Universal Robots PolyScope program: Main_JF.urp

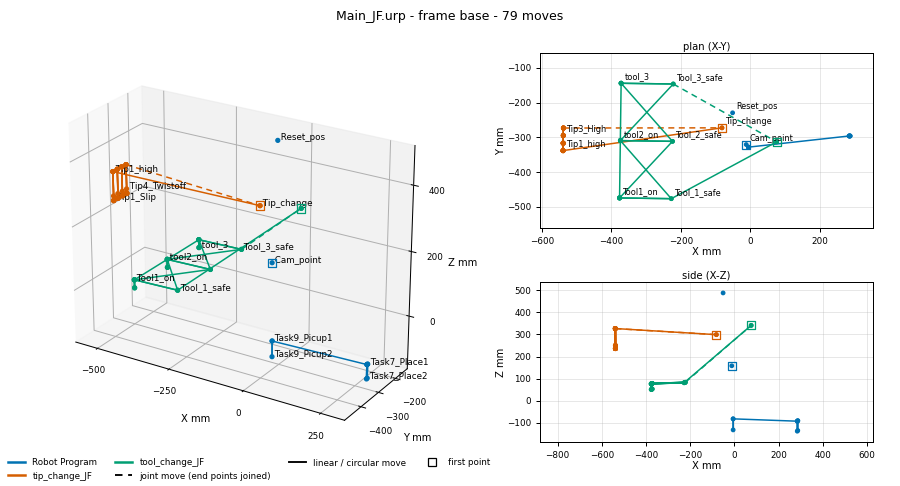
[picture p0: tool path of Main_JF.urp in frame base, 79 of 86 moves have a stored position in this frame; points joined in program order, loops and branches not executed]
Program Main_JF (installation=default directory=/programs/usbdisk/Billeder fra kamera createdIn=3.7.0.40195 lastSavedIn=3.10.1.76190 robotSerialNumber=2018359886)
Calibrated DH parameters: a=[-0.000111, -0.180064, -0.391564, 0.000025, 0.000035, 0]; d=[0.089308, 162.079685, -160.155007, -1.814221, 0.094754, 0.082578]; alpha=[1.569707, -0.002379, 0.010338, 1.570474, -1.569894, 0]; deltaTheta=[0.000021, -1.133914, 1.184629, -0.050828, 0.000017, 0.000075]
BeforeStart
  open := socket_open("192.168.0.15",30002)
  Old_Tool := 0
  Old_tip := 0
  Set DigitalOutput pin=config_out[4]; digitalValue=0
  Set DigitalOutput pin=config_out[5]; digitalValue=0
  Set DigitalOutput pin=config_out[6]; digitalValue=0
  Set DigitalOutput pin=config_out[7]; digitalValue=0
  Set DigitalOutput pin=config_out[0]; digitalValue=1
  Set DigitalOutput pin=config_out[2]; digitalValue=1
  Call Tool_initiation_tjeck
Robot Program (runOnlyOnce=false)
  Loop While (checkContinuously=false) expression=open≟ False
    open := socket_open("192.168.0.15",30002)
    Wait Sleep waitTime=0.5
  data := socket_read_ascii_float(8)
  Wait Sleep waitTime=0.5
  If data[0]≠0
    task := data[1]
    New_Tool_Setup := data[2]
    X_axis := data[3]
    Y_axis := data[4]
    Z_axis := data[5]
    X_rot := data[6]
    Y_rot := data[7]
    Z_rot := data[8]
    Rot := [d2r(data[6]),d2r(data[7]),d2r(data[8])]
    rot_v := rpy2rotvec(Rot)
    Insect_pos_High := p[X_axis,Y_axis,Z_axis+0.05,rot_v[0],rot_v[1],rot_v[2]]
    Insect_pos := p[X_axis,Y_axis,Z_axis,rot_v[0],rot_v[1],rot_v[2]]
    If New_Tool_Setup≠0
      If New_Tool_Setup>3
        New_tip := New_Tool_Setup-1
        New_Tool := 1
        Set NoAction tcp=TCP_Tips
      Else 
        New_tip := 0
        New_Tool := New_Tool_Setup
    Else 
      New_Tool := 0
      New_tip := 0
    If Old_Tool≟1 and New_tip≠Old_tip
      Call tip_change_JF
    SuppressedNode
      Switch expression=New_Tool
        Case (caseValue=1)
          Set NoAction tcp=TCP_Tool1
        Case (caseValue=2)
          Set NoAction tcp=TCP_Tool2
        Case (caseValue=3)
          Set NoAction tcp=TCP_Tool3
    If New_Tool≠Old_Tool
      Call tool_change_JF
    If New_tip≠Old_tip
      Call tip_change_JF
    SuppressedNode
      If New_tip≠Old_tip
        Popup Message (haltProgram=false message=Mount the correct tool tip. inputType=Text)
        Old_tip := New_tip
    If task≟1
      Wait Sleep waitTime=0.5
      Set SingleDigitalPulseActionState SingleDigitalPulseActionState(hiPulseInSeconds=0.5, pin=config_out[4])
      Set SingleDigitalPulseActionState SingleDigitalPulseActionState(hiPulseInSeconds=0.5, pin=config_out[5])
      Set SingleDigitalPulseActionState SingleDigitalPulseActionState(hiPulseInSeconds=0.5, pin=config_out[6])
      Set SingleDigitalPulseActionState SingleDigitalPulseActionState(hiPulseInSeconds=0.5, pin=config_out[7])
      Wait AnalogInput pin=analog_in[0]; analogComparison=0; analogValue=4
      Wait Sleep waitTime=0.5
      MoveL speed 250 mm/s, acceleration 1200 mm/s^2 (useActiveTCP=false) tcp=TCP_Cam; feature=Base
        SuppressedNode
          Waypoint ST_0_pos: TCP in base x=-75.138 y=-256.156 z=-140.441 mm, rx=0.4782 ry=3.0882 rz=0.0296 rad; joints [-83.913, -73.866, -152.197, -44.779, -268.413, 24.148] deg; flange x=-80.553 y=-258.226 z=132.545 mm, rx=0.4782 ry=3.0882 rz=0.0296 rad
        Waypoint Cam_point: TCP in base x=-11.711 y=-320.976 z=158.38 mm, rx=-0.0005 ry=-0.0003 rz=-3.1411 rad; joints [-100.01, -73.764, -127.296, -67.748, 91.294, -10.022] deg; flange x=-166.479 y=-319.785 z=277.387 mm, rx=-0.0077 ry=3.1318 rz=-0.0369 rad
        Wait Sleep waitTime=12
        SuppressedNode
          Waypoint Waypoint_1 (Relative): TCP in base x=286.294 y=-286.187 z=165.302 mm, rx=-0.0004 ry=0.0004 rz=3.1278 rad; joints [-44.345, -64.751, -131.64, -72.299, -270.032, 46.416] deg; flange x=131.485 y=-282.783 z=284.213 mm, rx=0.0146 ry=3.1313 rz=-0.0371 rad
    If task≟2
      Wait Sleep waitTime=0.5
      Set SingleDigitalPulseActionState SingleDigitalPulseActionState(hiPulseInSeconds=0.5, pin=config_out[4])
      Set SingleDigitalPulseActionState SingleDigitalPulseActionState(hiPulseInSeconds=0.5, pin=config_out[5])
      Set SingleDigitalPulseActionState SingleDigitalPulseActionState(hiPulseInSeconds=0.5, pin=config_out[6])
      Set SingleDigitalPulseActionState SingleDigitalPulseActionState(hiPulseInSeconds=0.5, pin=config_out[7])
      Wait AnalogInput pin=analog_in[0]; analogComparison=0; analogValue=4
      Wait Sleep waitTime=0.5
    If task≟3
      Wait Sleep waitTime=0.5
      Set SingleDigitalPulseActionState SingleDigitalPulseActionState(hiPulseInSeconds=0.5, pin=config_out[6])
      Set SingleDigitalPulseActionState SingleDigitalPulseActionState(hiPulseInSeconds=0.5, pin=config_out[7])
      Wait AnalogInput pin=analog_in[0]; analogComparison=0; analogValue=4
      Wait Sleep waitTime=0.5
    If task≟4
      Wait Sleep waitTime=0.5
      Set SingleDigitalPulseActionState SingleDigitalPulseActionState(hiPulseInSeconds=0.5, pin=config_out[4])
      Set SingleDigitalPulseActionState SingleDigitalPulseActionState(hiPulseInSeconds=0.5, pin=config_out[6])
      Set SingleDigitalPulseActionState SingleDigitalPulseActionState(hiPulseInSeconds=0.5, pin=config_out[7])
      Wait AnalogInput pin=analog_in[0]; analogComparison=0; analogValue=4
      Wait Sleep waitTime=0.5
    If task≟5
      Wait Sleep waitTime=0.5
      Set SingleDigitalPulseActionState SingleDigitalPulseActionState(hiPulseInSeconds=0.5, pin=config_out[5])
      Set SingleDigitalPulseActionState SingleDigitalPulseActionState(hiPulseInSeconds=0.5, pin=config_out[6])
      Set SingleDigitalPulseActionState SingleDigitalPulseActionState(hiPulseInSeconds=0.5, pin=config_out[7])
      Wait AnalogInput pin=analog_in[0]; analogComparison=0; analogValue=4
      Wait Sleep waitTime=0.5
    If task≟6
      Wait Sleep waitTime=0.5
      Set SingleDigitalPulseActionState SingleDigitalPulseActionState(hiPulseInSeconds=0.5, pin=config_out[4])
      Wait AnalogInput pin=analog_in[0]; analogComparison=0; analogValue=4
      Wait Sleep waitTime=0.5
      Set SingleDigitalPulseActionState SingleDigitalPulseActionState(hiPulseInSeconds=0.5, pin=config_out[5])
      Wait AnalogInput pin=analog_in[0]; analogComparison=0; analogValue=4
      Wait Sleep waitTime=0.5
    If task≟7
      Wait Sleep waitTime=0.5
      If New_Tool_Setup≟1
        Set NoAction tcp=TCP_Tool1
      Else 
        Set NoAction tcp=TCP_Tips
      MoveL speed 250 mm/s, acceleration 1200 mm/s^2 (useActiveTCP=true) feature=Base
        SuppressedNode
          Waypoint Task7_Picup1: TCP in base x=-2.957 y=-327.485 z=-88.615 mm, rx=-0.0002 ry=-0.0001 rz=1.5744 rad; joints [-84.172, -77.712, -147.228, -41.841, -255.532, 22.481] deg; flange x=-59.467 y=-294.342 z=154.237 mm, rx=0.3968 ry=2.8622 rz=0.009 rad
        SuppressedNode
          Waypoint Task7_Picup2: TCP in base x=-2.9 y=-327.528 z=-136.598 mm, rx=-0.0002 ry=0 rz=1.5745 rad; joints [-84.173, -87.531, -150.911, -28.32, -255.654, 22.544] deg; flange x=-59.407 y=-294.371 z=106.252 mm, rx=0.3967 ry=2.8623 rz=0.0089 rad
        Waypoint Waypoint (Variable): variable=Insect_pos_High
        SuppressedNode
          Waypoint Waypoint (Variable): variable=Insect_pos
      Set SingleDigitalPulseActionState SingleDigitalPulseActionState(hiPulseInSeconds=0.5, pin=config_out[6])
      Wait AnalogInput pin=analog_in[0]; analogComparison=0; analogValue=4
      MoveL speed 250 mm/s, acceleration 1200 mm/s^2 (useActiveTCP=true) feature=Base
        Waypoint Waypoint (Variable): variable=Insect_pos
      Set SingleDigitalPulseActionState SingleDigitalPulseActionState(hiPulseInSeconds=0.5, pin=config_out[5])
      Set SingleDigitalPulseActionState SingleDigitalPulseActionState(hiPulseInSeconds=0.5, pin=config_out[6])
      Wait AnalogInput pin=analog_in[0]; analogComparison=0; analogValue=4
      Wait Sleep waitTime=0.5
      MoveL speed 250 mm/s, acceleration 1200 mm/s^2 (useActiveTCP=true) feature=Base
        SuppressedNode
          Waypoint Task7_Picup1: TCP in base x=-2.957 y=-327.485 z=-88.615 mm, rx=-0.0002 ry=-0.0001 rz=1.5744 rad; joints [-84.172, -77.712, -147.228, -41.841, -255.532, 22.481] deg; flange x=-59.467 y=-294.342 z=154.237 mm, rx=0.3968 ry=2.8622 rz=0.009 rad
        Waypoint Waypoint (Variable): variable=Insect_pos_High
        Waypoint Task7_Place1: TCP in base x=286.894 y=-296.293 z=-90.183 mm, rx=-0.0001 ry=0.0004 rz=0.0005 rad; joints [-32.091, -86.998, -142.363, -29.578, 96.187, 74.653] deg; flange x=236.868 y=-267.234 z=154.959 mm, rx=0.3978 ry=2.8963 rz=0.0236 rad
        Waypoint Task7_Place2: TCP in base x=286.843 y=-296.296 z=-134.286 mm, rx=-0.0001 ry=0.0005 rz=0.0005 rad; joints [-32.094, -95.154, -145.064, -18.726, 96.08, 74.681] deg; flange x=236.849 y=-267.236 z=110.862 mm, rx=0.3978 ry=2.8964 rz=0.0236 rad
      Set SingleDigitalPulseActionState SingleDigitalPulseActionState(hiPulseInSeconds=0.5, pin=config_out[4])
      Set SingleDigitalPulseActionState SingleDigitalPulseActionState(hiPulseInSeconds=0.5, pin=config_out[5])
      Wait AnalogInput pin=analog_in[0]; analogComparison=0; analogValue=4
      Wait Sleep waitTime=0.5
      MoveL speed 250 mm/s, acceleration 1200 mm/s^2 (useActiveTCP=true) feature=Base
        Waypoint Task7_Place1: TCP in base x=286.894 y=-296.293 z=-90.183 mm, rx=-0.0001 ry=0.0004 rz=0.0005 rad; joints [-32.091, -86.998, -142.363, -29.578, 96.187, 74.653] deg; flange x=236.868 y=-267.234 z=154.959 mm, rx=0.3978 ry=2.8963 rz=0.0236 rad
      Wait Sleep waitTime=0.5
    If task≟8
      Wait Sleep waitTime=0.5
      Set AnalogOutput pin=analog_out[0]; analogValue=10
      Set AnalogOutput pin=analog_out[1]; analogValue=8
      MoveL speed 250 mm/s, acceleration 1200 mm/s^2 (useActiveTCP=false) tcp=TCP_Tool2; feature=Base
        SuppressedNode
          Waypoint Task8_Picup1: TCP in base x=-2.943 y=-327.466 z=-88.616 mm, rx=-0.006 ry=3.1413 rz=-0.0002 rad; joints [-71.062, -76.126, -140.922, -52.984, -269.542, 19.116] deg; flange x=-3.919 y=-325.243 z=184.421 mm, rx=-0.006 ry=3.1413 rz=-0.0002 rad
        Waypoint Waypoint (Variable): variable=Insect_pos_High
      Set SingleDigitalPulseActionState SingleDigitalPulseActionState(hiPulseInSeconds=2.5, pin=digital_out[2])
      Wait Sleep waitTime=2.5
      MoveL speed 250 mm/s, acceleration 1200 mm/s^2 (useActiveTCP=false) tcp=TCP_Tool2; feature=Base
        SuppressedNode
          Waypoint Task8_Picup2: TCP in base x=-2.923 y=-327.461 z=-138.602 mm, rx=-0.0059 ry=3.1414 rz=-0.0002 rad; joints [-71.069, -83.732, -145.267, -41.035, -269.637, 19.19] deg; flange x=-3.873 y=-325.242 z=134.435 mm, rx=-0.0059 ry=3.1414 rz=-0.0002 rad
        Waypoint Waypoint (Variable): variable=Insect_pos
      Set SingleDigitalPulseActionState SingleDigitalPulseActionState(hiPulseInSeconds=2.5, pin=digital_out[1])
      Wait Sleep waitTime=2.5
      MoveL speed 250 mm/s, acceleration 1200 mm/s^2 (useActiveTCP=false) tcp=TCP_Tool2; feature=Base
        SuppressedNode
          Waypoint Task8_Picup1: TCP in base x=-2.943 y=-327.466 z=-88.616 mm, rx=-0.006 ry=3.1413 rz=-0.0002 rad; joints [-71.062, -76.126, -140.922, -52.984, -269.542, 19.116] deg; flange x=-3.919 y=-325.243 z=184.421 mm, rx=-0.006 ry=3.1413 rz=-0.0002 rad
        Waypoint Waypoint (Variable): variable=Insect_pos_High
        Waypoint Task8_Place1: TCP in base x=284.494 y=-296.271 z=-92.185 mm, rx=-0.0002 ry=-0.0002 rz=0.0035 rad; joints [-30.716, -90.016, -130.004, -50.01, 90.403, 59.471] deg; flange x=284.456 y=-296.209 z=180.855 mm, rx=-0.0057 ry=3.1414 rz=-0.0004 rad
        Waypoint Task8_Place2: TCP in base x=284.497 y=-296.263 z=-137.47 mm, rx=-0.0002 ry=-0.0002 rz=0.0037 rad; joints [-30.723, -95.697, -133.143, -41.191, 90.336, 59.513] deg; flange x=284.465 y=-296.198 z=135.57 mm, rx=-0.0058 ry=3.1415 rz=-0.0004 rad
      Set SingleDigitalPulseActionState SingleDigitalPulseActionState(hiPulseInSeconds=2.5, pin=digital_out[2])
      Wait Sleep waitTime=2.5
      MoveL speed 250 mm/s, acceleration 1200 mm/s^2 (useActiveTCP=false) tcp=TCP_Tool2; feature=Base
        Waypoint Task8_Place1: TCP in base x=284.494 y=-296.271 z=-92.185 mm, rx=-0.0002 ry=-0.0002 rz=0.0035 rad; joints [-30.716, -90.016, -130.004, -50.01, 90.403, 59.471] deg; flange x=284.456 y=-296.209 z=180.855 mm, rx=-0.0057 ry=3.1414 rz=-0.0004 rad
      Wait Sleep waitTime=0.5
    If task≟9
      Wait Sleep waitTime=0.5
      Set DigitalOutput pin=digital_out[3]; digitalValue=1
      Set SingleDigitalPulseActionState SingleDigitalPulseActionState(hiPulseInSeconds=0.2, pin=digital_out[4])
      Wait Sleep waitTime=0.5
      MoveL speed 250 mm/s, acceleration 1200 mm/s^2 (useActiveTCP=false) tcp=TCP_Tool3; feature=Base
        Waypoint Task9_Picup1: TCP in base x=-5.553 y=-328.417 z=-81.63 mm, rx=-0.0001 ry=0 rz=-0.2794 rad; joints [-71.641, -82.877, -143.87, -43.297, 90.369, 34.822] deg; flange x=-5.553 y=-330.02 z=144.05 mm, rx=-0.4373 ry=-3.111 rz=0 rad
        Waypoint Task9_Picup2: TCP in base x=-5.569 y=-328.42 z=-131.615 mm, rx=-0.0002 ry=-0.0001 rz=-0.2795 rad; joints [-71.657, -92.36, -147.267, -30.41, 90.258, 34.878] deg; flange x=-5.583 y=-329.999 z=94.065 mm, rx=0.4375 ry=3.111 rz=-0.0002 rad
      Set SingleDigitalPulseActionState SingleDigitalPulseActionState(hiPulseInSeconds=0.2, pin=digital_out[5])
      Wait Sleep waitTime=0.5
      MoveL speed 250 mm/s, acceleration 1200 mm/s^2 (useActiveTCP=false) tcp=TCP_Tool3; feature=Base
        Waypoint Task9_Picup1: TCP in base x=-5.553 y=-328.417 z=-81.63 mm, rx=-0.0001 ry=0 rz=-0.2794 rad; joints [-71.641, -82.877, -143.87, -43.297, 90.369, 34.822] deg; flange x=-5.553 y=-330.02 z=144.05 mm, rx=-0.4373 ry=-3.111 rz=0 rad
      Set DigitalOutput pin=digital_out[3]; digitalValue=0
      Wait Sleep waitTime=0.5
    If task≟10
      Wait Sleep waitTime=0.5
      If New_Tool≟1
        Set NoAction tcp=TCP_Tool1
      If New_Tool≟2
        Set NoAction tcp=TCP_Tool2
      If New_Tool≟3
        Set NoAction tcp=TCP_Tool3
      If New_tip≠0
        Set NoAction tcp=TCP_Tips
      Wait Sleep waitTime=0.5
      MoveL speed 250 mm/s, acceleration 1200 mm/s^2 (useActiveTCP=true) feature=Base
        Waypoint Waypoint (Variable): variable=Insect_pos
      Wait Sleep waitTime=0.5
    If task≟55
      MoveJ speed 60 deg/s, acceleration 80 deg/s^2 (useActiveTCP=false) tcp=TCP_Schunk
        Waypoint Reset_pos: TCP in base x=-50.952 y=-229.593 z=487.929 mm, rx=-0.1979 ry=-0.2122 rz=-1.8134 rad; joints [-70.558, -50.466, -101.852, -104.572, 84.568, 123.197] deg; flange x=-49.676 y=-215.711 z=542.145 mm, rx=2.3303 ry=1.8037 rz=-0.2542 rad
      Script: socket_send_string("Done")
      Popup Message (haltProgram=true message=Labview stopped inputType=Text)
    SuppressedNode
      pos_calc := p[pos_raw[1]/1000,pos_raw[2]/1000,pos_raw[3]/1000,d2r(pos_raw[4]),d2r(pos_raw[5]),d2r(pos_raw[6])]
    SuppressedNode
      act_pos := get_actual_tcp_pose()
    SuppressedNode
      transfer := pose_trans(act_pos,pos_calc)
    SuppressedNode
      MoveJ speed 60 deg/s, acceleration 80 deg/s^2 (useActiveTCP=true)
        Waypoint Waypoint (Variable): variable=pos_calc
        Wait Sleep waitTime=1
        SuppressedNode
          Waypoint pos_init: TCP in base x=-499.955 y=-310.203 z=526.258 mm, rx=1.0312 ry=1.3413 rz=-1.0697 rad; joints [12.579, -80.638, 78.252, -89.492, -0.093, -0.387] deg
    SuppressedNode
      Script: socket_send_string("Done")
    SuppressedNode
      Script: socket_close()
  Script: socket_send_string("Done")
SubProgram -> Tool_initiation_tjeck
SubProgram -> tool_change_JF
SubProgram -> tip_change_JF
SubProgram Tool_initiation_tjeck (keepSynchronizedWithDisk=false trackProgramExecution=true) programFile=/programs/Tool initiation tjeck.urp
  Active_tools := 0
  If digital_in[4]≟ False
    Old_Tool := 1
    Active_tools := Active_tools+1
    Set DigitalOutput tcp=TCP_Tool1; pin=digital_out[6]; digitalValue=1
    SuppressedNode
      Popup Message (haltProgram=false message=Tool 1 active inputType=Text)
  If digital_in[5]≟ False
    Old_Tool := 2
    Active_tools := Active_tools+1
    Set DigitalOutput tcp=TCP_Tool2; pin=digital_out[6]; digitalValue=1
    SuppressedNode
      Popup Message (haltProgram=false message=Tool 2 active inputType=Text)
  If digital_in[6]≟ False
    Old_Tool := 3
    Active_tools := Active_tools+1
    Set DigitalOutput tcp=TCP_Tool3; pin=digital_out[6]; digitalValue=1
    SuppressedNode
      Popup Message (haltProgram=false message=Tool 3 active inputType=Text)
  If digital_in[4] and digital_in[5] and digital_in[6]≟ True
    Old_Tool := 0
    SuppressedNode
      Popup Message (haltProgram=false message=Tool 0 active inputType=Text)
  If Active_tools>1
    Popup Message (haltProgram=false message=Reset Tools inputType=Text)
  SuppressedNode
    Wait Sleep waitTime=5
SubProgram tip_change_JF (keepSynchronizedWithDisk=true trackProgramExecution=false) programFile=/programs/tip_change_JF.urp
  MoveJ speed 60 deg/s, acceleration 80 deg/s^2 (useActiveTCP=false) tcp=TCP_Tool1
    Waypoint Tip_change: TCP in base x=-81.571 y=-272.848 z=299.256 mm, rx=0 ry=0.0001 rz=-1.545 rad; joints [-70.556, -50.466, -101.854, -104.569, 84.569, 123.199] deg; flange x=-49.667 y=-215.719 z=542.134 mm, rx=2.3303 ry=1.8037 rz=-0.2542 rad
  Set NoAction tcp=TCP_Tool1
  'skipping tip 0-> No tool on robot'
  If Old_tip≟3
    MoveL speed 250 mm/s, acceleration 1200 mm/s^2 (useActiveTCP=false) tcp=TCP_Tool1; feature=Joint_6_name
      Waypoint Tip1_high: TCP in base x=-538.968 y=-338.378 z=326.942 mm, rx=-0.0068 ry=0.0085 rz=3.1265 rad; joints [-131.445, -107.957, -50.262, -104.103, 80.885, 154.293] deg; pose in feature x=57.214 y=-30.744 z=76.425 mm, rx=0 ry=0.0001 rz=-2.0641 rad; flange x=-490.354 y=-366.84 z=572.437 mm, rx=3.0721 ry=-0.4473 rz=-0.3327 rad
      Waypoint Tip1_Slip: TCP in base x=-538.568 y=-337.869 z=236.939 mm, rx=-0.0068 ry=0.0085 rz=3.1242 rad; joints [-131.488, -104.349, -68.619, -89.398, 80.899, 154.544] deg; pose in feature x=-140.414 y=-433.139 z=348.51 mm, rx=0.0255 ry=-0.0126 rz=-1.9429 rad; flange x=-490.024 y=-366.448 z=482.434 mm, rx=3.0718 ry=-0.4509 rz=-0.3328 rad
      Waypoint Tip1_Lock: TCP in base x=-538.583 y=-338.869 z=236.944 mm, rx=0.0013 ry=-0.0083 rz=-2.1118 rad; joints [-137.124, -99.221, -76.057, -82.468, 93.606, 89.965] deg; pose in feature x=-139.482 y=-433.5 z=348.531 mm, rx=0.0139 ry=-0.0208 rz=-0.8958 rad; flange x=-488.924 y=-309.541 z=482.128 mm, rx=2.7896 ry=1.107 rz=-0.2715 rad
      Waypoint Tip1_Twistoff: TCP in base x=-538.643 y=-338.793 z=250.944 mm, rx=-0.0027 ry=-0.0068 rz=-1.059 rad; joints [-143.816, -105.991, -63.242, -98.539, 103.242, 22.663] deg; pose in feature x=-0.02 y=-0.021 z=11.036 mm, rx=-0.0001 ry=0 rz=1.0527 rad; flange x=-538.901 y=-279.541 z=495.751 mm, rx=1.814 ry=2.3069 rz=-0.1444 rad
      Waypoint Tip1_high: TCP in base x=-538.968 y=-338.378 z=326.942 mm, rx=-0.0068 ry=0.0085 rz=3.1265 rad; joints [-131.445, -107.957, -50.262, -104.103, 80.885, 154.293] deg; pose in feature x=57.214 y=-30.744 z=76.425 mm, rx=0 ry=0.0001 rz=-2.0641 rad; flange x=-490.354 y=-366.84 z=572.437 mm, rx=3.0721 ry=-0.4473 rz=-0.3327 rad
    SuppressedNode
      MoveL speed 250 mm/s, acceleration 1200 mm/s^2 (useActiveTCP=false) tcp=TCP_Tool1; feature=Joint_6_name
        Waypoint Tip1_high: TCP in base x=-537.538 y=-337.809 z=326.901 mm, rx=0.0003 ry=0.0002 rz=-1.5826 rad; joints [-130.16, -106.928, -52.243, -102.922, -281.606, 155.501] deg; pose in feature x=0.604 y=0.279 z=0.912 mm, rx=0 ry=0.0001 rz=0.0099 rad; flange x=-481.613 y=-371.883 z=569.759 mm, rx=3.08 ry=-0.4512 rz=-0.394 rad
        Waypoint Tip1_press: TCP in base x=-537.53 y=-337.783 z=237.901 mm, rx=0.0003 ry=0 rz=-0.5354 rad; joints [-136.639, -97.589, -78.691, -79.527, -267.198, 90.394] deg; pose in feature x=-0.011 y=0.014 z=-89.017 mm, rx=0 ry=-0.0001 rz=1.0471 rad; flange x=-480.131 y=-306.405 z=480.779 mm, rx=2.7834 ry=1.1057 rz=-0.3248 rad
        Waypoint Tip1_Lock: TCP in base x=-537.531 y=-337.784 z=239.901 mm, rx=0.0003 ry=0 rz=-0.5354 rad; joints [-136.638, -97.608, -78.375, -79.823, -267.198, 90.392] deg; pose in feature x=-0.011 y=0.014 z=-87.017 mm, rx=0 ry=0 rz=1.0471 rad; flange x=-480.132 y=-306.408 z=482.779 mm, rx=2.7834 ry=1.1057 rz=-0.3248 rad
        Waypoint Tip1_Slip: TCP in base x=-537.531 y=-337.783 z=238.901 mm, rx=0.0003 ry=0.0001 rz=-1.5826 rad; joints [-130.205, -103.681, -69.728, -88.707, -281.576, 155.612] deg; pose in feature x=0.094 y=0.018 z=1.031 mm, rx=-0.0001 ry=-0.0001 rz=0.0001 rad; flange x=-481.61 y=-371.853 z=481.761 mm, rx=3.0799 ry=-0.4512 rz=-0.3939 rad
        Waypoint Tip1_high: TCP in base x=-537.538 y=-337.809 z=326.901 mm, rx=0.0003 ry=0.0002 rz=-1.5826 rad; joints [-130.16, -106.928, -52.243, -102.922, -281.606, 155.501] deg; pose in feature x=0.604 y=0.279 z=0.912 mm, rx=0 ry=0.0001 rz=0.0099 rad; flange x=-481.613 y=-371.883 z=569.759 mm, rx=3.08 ry=-0.4512 rz=-0.394 rad
  If Old_tip≟4
    MoveL speed 250 mm/s, acceleration 1200 mm/s^2 (useActiveTCP=false) tcp=TCP_Tool1; feature=Joint_6_name
      Waypoint Tip2_High: TCP in base x=-538.644 y=-316.88 z=326.826 mm, rx=-0.0068 ry=0.0085 rz=3.1265 rad; joints [-132.848, -105.784, -53.248, -103.06, 81.079, 152.898] deg; pose in feature x=2.19 y=1.693 z=81.747 mm, rx=-0.0035 ry=0.0068 rz=-0.958 rad; flange x=-490.029 y=-345.343 z=572.321 mm, rx=3.0721 ry=-0.4473 rz=-0.3327 rad
      Waypoint Tip2_Slip: TCP in base x=-538.244 y=-316.372 z=236.823 mm, rx=-0.0068 ry=0.0085 rz=3.1265 rad; joints [-132.898, -102.409, -71.128, -88.573, 81.109, 153.006] deg; pose in feature x=-160.454 y=-425.366 z=348.057 mm, rx=0.0255 ry=-0.0126 rz=-1.9406 rad; flange x=-489.629 y=-344.835 z=482.318 mm, rx=3.0721 ry=-0.4473 rz=-0.3327 rad
      Waypoint Tip2_Lock: TCP in base x=-538.259 y=-317.372 z=236.828 mm, rx=0.0012 ry=-0.0083 rz=-2.1095 rad; joints [-138.801, -97.64, -77.885, -82.321, 93.99, 88.197] deg; pose in feature x=-159.522 y=-425.727 z=348.078 mm, rx=0.0138 ry=-0.0208 rz=-0.8934 rad; flange x=-488.666 y=-287.924 z=482.011 mm, rx=2.7881 ry=1.1102 rz=-0.2712 rad
      Waypoint Tip2_Twistoff: TCP in base x=-538.319 y=-317.295 z=250.828 mm, rx=-0.0027 ry=-0.0068 rz=-1.0623 rad; joints [-145.487, -104.574, -65.006, -98.529, 103.298, 21.145] deg; pose in feature x=-0.013 y=0.071 z=-74.909 mm, rx=0.0001 ry=-0.0001 rz=2.0945 rad; flange x=-538.389 y=-258.046 z=495.635 mm, rx=1.8178 ry=2.3041 rz=-0.1448 rad
      Waypoint Tip2_High: TCP in base x=-538.644 y=-316.88 z=326.826 mm, rx=-0.0068 ry=0.0085 rz=3.1265 rad; joints [-132.848, -105.784, -53.248, -103.06, 81.079, 152.898] deg; pose in feature x=2.19 y=1.693 z=81.747 mm, rx=-0.0035 ry=0.0068 rz=-0.958 rad; flange x=-490.029 y=-345.343 z=572.321 mm, rx=3.0721 ry=-0.4473 rz=-0.3327 rad
    SuppressedNode
      MoveL speed 250 mm/s, acceleration 1200 mm/s^2 (useActiveTCP=false) tcp=TCP_Tool1; feature=Joint_6_name
        Waypoint Tip2_High: TCP in base x=-537.283 y=-316.311 z=326.907 mm, rx=0.0003 ry=0.0002 rz=-1.5826 rad; joints [-131.544, -104.755, -55.177, -101.873, -281.409, 154.115] deg; pose in feature x=-21.513 y=0.011 z=-0.018 mm, rx=0 ry=0 rz=-0.0001 rad; flange x=-481.359 y=-350.384 z=569.766 mm, rx=3.08 ry=-0.4512 rz=-0.394 rad
        Waypoint Tip2_Press: TCP in base x=-537.276 y=-316.285 z=237.907 mm, rx=0.0003 ry=0 rz=-0.5354 rad; joints [-138.326, -96.017, -80.448, -79.412, -266.784, 88.762] deg; pose in feature x=-21.511 y=0.015 z=-89.018 mm, rx=0 ry=-0.0001 rz=1.0471 rad; flange x=-479.877 y=-284.907 z=480.785 mm, rx=2.7834 ry=1.1057 rz=-0.3248 rad
        Waypoint Tip2_Lock: TCP in base x=-537.276 y=-316.285 z=239.907 mm, rx=0.0003 ry=0 rz=-0.5354 rad; joints [-138.325, -96.035, -80.135, -79.708, -266.784, 88.759] deg; pose in feature x=-21.511 y=0.015 z=-87.018 mm, rx=0 ry=0 rz=1.0471 rad; flange x=-479.878 y=-284.909 z=482.785 mm, rx=2.7834 ry=1.1057 rz=-0.3248 rad
        Waypoint Tip2_Slip: TCP in base x=-537.276 y=-316.285 z=238.907 mm, rx=0.0003 ry=0.0001 rz=-1.5826 rad; joints [-131.59, -101.734, -72.212, -87.881, -281.381, 154.223] deg; pose in feature x=-21.511 y=0.015 z=-88.018 mm, rx=0.0001 ry=0 rz=-0.0001 rad; flange x=-481.356 y=-350.354 z=481.767 mm, rx=3.0799 ry=-0.4512 rz=-0.3939 rad
        Waypoint Tip2_High: TCP in base x=-537.283 y=-316.311 z=326.907 mm, rx=0.0003 ry=0.0002 rz=-1.5826 rad; joints [-131.544, -104.755, -55.177, -101.873, -281.409, 154.115] deg; pose in feature x=-21.513 y=0.011 z=-0.018 mm, rx=0 ry=0 rz=-0.0001 rad; flange x=-481.359 y=-350.384 z=569.766 mm, rx=3.08 ry=-0.4512 rz=-0.394 rad
  If Old_tip≟5
    MoveL speed 250 mm/s, acceleration 1200 mm/s^2 (useActiveTCP=false) tcp=TCP_Tool1; feature=Joint_6_name
      Waypoint Tip3_High: TCP in base x=-538.312 y=-294.883 z=326.707 mm, rx=-0.0068 ry=0.0085 rz=3.1265 rad; joints [-134.359, -103.714, -56.012, -102.124, 81.293, 151.396] deg; pose in feature x=13.69 y=-3.755 z=-38.348 mm, rx=-0.1637 ry=0.1574 rz=-0.0025 rad; flange x=-489.697 y=-323.346 z=572.202 mm, rx=3.0721 ry=-0.4473 rz=-0.3327 rad
      Waypoint Tip3_Slip: TCP in base x=-537.912 y=-294.375 z=236.704 mm, rx=-0.0068 ry=0.0085 rz=3.1265 rad; joints [-134.411, -100.547, -73.471, -87.848, 81.321, 151.499] deg; pose in feature x=-180.961 y=-417.412 z=347.593 mm, rx=0.0255 ry=-0.0126 rz=-1.9406 rad; flange x=-489.297 y=-322.838 z=482.199 mm, rx=3.0721 ry=-0.4473 rz=-0.3327 rad
      Waypoint Tip3_Lock: TCP in base x=-537.927 y=-295.375 z=236.709 mm, rx=0.0012 ry=-0.0083 rz=-2.1095 rad; joints [-140.58, -96.119, -79.595, -82.242, 94.365, 86.458] deg; pose in feature x=-180.029 y=-417.773 z=347.614 mm, rx=0.0138 ry=-0.0208 rz=-0.8934 rad; flange x=-488.334 y=-265.927 z=481.892 mm, rx=2.7881 ry=1.1102 rz=-0.2712 rad
      Waypoint Tip3_Twistoff: TCP in base x=-537.987 y=-295.298 z=250.709 mm, rx=-0.0027 ry=-0.0068 rz=-1.0623 rad; joints [-147.274, -103.276, -66.568, -98.672, 103.353, 19.316] deg; pose in feature x=-1.767 y=-0.914 z=5.336 mm, rx=0 ry=0 rz=1.0005 rad; flange x=-538.057 y=-236.049 z=495.517 mm, rx=1.8178 ry=2.3041 rz=-0.1448 rad
      Waypoint Tip3_High: TCP in base x=-538.312 y=-294.883 z=326.707 mm, rx=-0.0068 ry=0.0085 rz=3.1265 rad; joints [-134.359, -103.714, -56.012, -102.124, 81.293, 151.396] deg; pose in feature x=13.69 y=-3.755 z=-38.348 mm, rx=-0.1637 ry=0.1574 rz=-0.0025 rad; flange x=-489.697 y=-323.346 z=572.202 mm, rx=3.0721 ry=-0.4473 rz=-0.3327 rad
    SuppressedNode
      MoveL speed 250 mm/s, acceleration 1200 mm/s^2 (useActiveTCP=false) tcp=TCP_Tool1; feature=Joint_6_name
        Waypoint Tip3_High: TCP in base x=-537.023 y=-294.313 z=326.914 mm, rx=0.0003 ry=0.0002 rz=-1.5826 rad; joints [-133.038, -102.675, -57.902, -100.922, -281.189, 152.62] deg; pose in feature x=-43.513 y=0.013 z=-0.018 mm, rx=0 ry=0 rz=-0.0001 rad; flange x=-481.098 y=-328.386 z=569.772 mm, rx=3.08 ry=-0.4512 rz=-0.394 rad
        Waypoint Tip3_Press: TCP in base x=-537.016 y=-294.286 z=237.914 mm, rx=0.0003 ry=0 rz=-0.5354 rad; joints [-140.139, -94.506, -82.089, -79.372, -266.341, 87.005] deg; pose in feature x=-43.511 y=0.017 z=-89.018 mm, rx=0 ry=-0.0001 rz=1.0471 rad; flange x=-479.616 y=-262.908 z=480.792 mm, rx=2.7834 ry=1.1057 rz=-0.3248 rad
        Waypoint Tip3_Lock: TCP in base x=-537.016 y=-294.287 z=239.914 mm, rx=0.0003 ry=0 rz=-0.5354 rad; joints [-140.138, -94.523, -81.777, -79.667, -266.341, 87.003] deg; pose in feature x=-43.511 y=0.016 z=-87.018 mm, rx=0 ry=0 rz=1.0471 rad; flange x=-479.617 y=-262.911 z=482.792 mm, rx=2.7834 ry=1.1057 rz=-0.3248 rad
        Waypoint Tip3_Slip: TCP in base x=-537.016 y=-294.286 z=238.914 mm, rx=0.0003 ry=0.0001 rz=-1.5826 rad; joints [-133.083, -99.839, -74.567, -87.115, -281.163, 152.725] deg; pose in feature x=-43.511 y=0.017 z=-88.018 mm, rx=0.0001 ry=0 rz=-0.0001 rad; flange x=-481.095 y=-328.356 z=481.774 mm, rx=3.0799 ry=-0.4512 rz=-0.3939 rad
        Waypoint Tip3_High: TCP in base x=-537.023 y=-294.313 z=326.914 mm, rx=0.0003 ry=0.0002 rz=-1.5826 rad; joints [-133.038, -102.675, -57.902, -100.922, -281.189, 152.62] deg; pose in feature x=-43.513 y=0.013 z=-0.018 mm, rx=0 ry=0 rz=-0.0001 rad; flange x=-481.098 y=-328.386 z=569.772 mm, rx=3.08 ry=-0.4512 rz=-0.394 rad
  If Old_tip≟6
    MoveL speed 250 mm/s, acceleration 1200 mm/s^2 (useActiveTCP=false) tcp=TCP_Tool1; feature=Joint_6_name
      Waypoint Tip4_High: TCP in base x=-537.988 y=-273.386 z=326.591 mm, rx=-0.0068 ry=0.0085 rz=3.1265 rad; joints [-135.913, -101.826, -58.462, -101.318, 81.519, 149.851] deg; pose in feature x=-0.038 y=0.033 z=76.429 mm, rx=0 ry=0.0001 rz=-2.0641 rad; flange x=-489.373 y=-301.849 z=572.086 mm, rx=3.0721 ry=-0.4473 rz=-0.3327 rad
      Waypoint Tip4_Slip: TCP in base x=-537.588 y=-272.878 z=236.588 mm, rx=-0.0068 ry=0.0085 rz=3.1265 rad; joints [-135.967, -98.824, -75.586, -87.211, 81.546, 149.951] deg; pose in feature x=-201.001 y=-409.638 z=347.14 mm, rx=0.0255 ry=-0.0126 rz=-1.9406 rad; flange x=-488.973 y=-301.34 z=482.083 mm, rx=3.0721 ry=-0.4473 rz=-0.3327 rad
      Waypoint Tip4_Lock: TCP in base x=-537.603 y=-273.877 z=236.593 mm, rx=0.0012 ry=-0.0083 rz=-2.1095 rad; joints [-142.401, -94.732, -81.112, -82.237, 94.745, 84.676] deg; pose in feature x=-200.069 y=-410 z=347.161 mm, rx=0.0138 ry=-0.0208 rz=-0.8934 rad; flange x=-488.01 y=-244.43 z=481.776 mm, rx=2.7881 ry=1.1102 rz=-0.2712 rad
      Waypoint Tip4_Twistoff: TCP in base x=-537.663 y=-273.801 z=250.593 mm, rx=-0.0027 ry=-0.0068 rz=-1.0623 rad; joints [-149.082, -102.119, -67.921, -98.888, 103.396, 17.462] deg; pose in feature x=-0.04 y=0.039 z=0.429 mm, rx=0.0001 ry=0 rz=0.0303 rad; flange x=-537.733 y=-214.552 z=495.401 mm, rx=1.8178 ry=2.3041 rz=-0.1448 rad
      Waypoint Tip4_High: TCP in base x=-537.988 y=-273.386 z=326.591 mm, rx=-0.0068 ry=0.0085 rz=3.1265 rad; joints [-135.913, -101.826, -58.462, -101.318, 81.519, 149.851] deg; pose in feature x=-0.038 y=0.033 z=76.429 mm, rx=0 ry=0.0001 rz=-2.0641 rad; flange x=-489.373 y=-301.849 z=572.086 mm, rx=3.0721 ry=-0.4473 rz=-0.3327 rad
    SuppressedNode
      MoveL speed 250 mm/s, acceleration 1200 mm/s^2 (useActiveTCP=false) tcp=TCP_Tool1; feature=Joint_6_name
        Waypoint Tip4_High: TCP in base x=-536.768 y=-272.814 z=326.92 mm, rx=0.0003 ry=0.0002 rz=-1.5826 rad; joints [-134.575, -100.773, -60.327, -100.092, -280.955, 151.081] deg; pose in feature x=-65.013 y=0.014 z=-0.019 mm, rx=0 ry=0 rz=-0.0001 rad; flange x=-480.844 y=-306.888 z=569.779 mm, rx=3.08 ry=-0.4512 rz=-0.394 rad
        Waypoint Tip4_Press: TCP in base x=-536.761 y=-272.788 z=237.92 mm, rx=0.0003 ry=0 rz=-0.5354 rad; joints [-141.998, -93.127, -83.542, -79.403, -265.89, 85.201] deg; pose in feature x=-65.011 y=0.018 z=-89.019 mm, rx=0 ry=-0.0001 rz=1.0471 rad; flange x=-479.362 y=-241.41 z=480.798 mm, rx=2.7834 ry=1.1057 rz=-0.3248 rad
        Waypoint Tip4_Lock: TCP in base x=-536.761 y=-272.788 z=239.92 mm, rx=0.0003 ry=0 rz=-0.5354 rad; joints [-141.997, -93.144, -83.231, -79.697, -265.89, 85.199] deg; pose in feature x=-65.011 y=0.018 z=-87.019 mm, rx=0 ry=0 rz=1.0471 rad; flange x=-479.363 y=-241.412 z=482.798 mm, rx=2.7834 ry=1.1057 rz=-0.3248 rad
        Waypoint Tip4_Slip: TCP in base x=-536.761 y=-272.788 z=238.92 mm, rx=0.0003 ry=0.0001 rz=-1.5826 rad; joints [-134.621, -98.08, -76.697, -86.434, -280.931, 151.185] deg; pose in feature x=-65.011 y=0.018 z=-88.019 mm, rx=0.0001 ry=0 rz=-0.0001 rad; flange x=-480.841 y=-306.857 z=481.78 mm, rx=3.0799 ry=-0.4512 rz=-0.3939 rad
        Waypoint Tip4_High: TCP in base x=-536.768 y=-272.814 z=326.92 mm, rx=0.0003 ry=0.0002 rz=-1.5826 rad; joints [-134.575, -100.773, -60.327, -100.092, -280.955, 151.081] deg; pose in feature x=-65.013 y=0.014 z=-0.019 mm, rx=0 ry=0 rz=-0.0001 rad; flange x=-480.844 y=-306.888 z=569.779 mm, rx=3.08 ry=-0.4512 rz=-0.394 rad
  If New_tip≟3
    MoveL speed 250 mm/s, acceleration 1200 mm/s^2 (useActiveTCP=false) tcp=TCP_Tool1; feature=Joint_6_name
      Waypoint Tip1_high: TCP in base x=-538.968 y=-338.378 z=326.942 mm, rx=-0.0068 ry=0.0085 rz=3.1265 rad; joints [-131.445, -107.957, -50.262, -104.103, 80.885, 154.293] deg; pose in feature x=57.214 y=-30.744 z=76.425 mm, rx=0 ry=0.0001 rz=-2.0641 rad; flange x=-490.354 y=-366.84 z=572.437 mm, rx=3.0721 ry=-0.4473 rz=-0.3327 rad
      Waypoint Tip1_press: TCP in base x=-538.579 y=-338.875 z=235.944 mm, rx=0.0013 ry=-0.0083 rz=-2.1118 rad; joints [-137.124, -99.209, -76.218, -82.319, 93.606, 89.967] deg; pose in feature x=-139.458 y=-433.497 z=347.532 mm, rx=0.0139 ry=-0.0208 rz=-0.8958 rad; flange x=-488.92 y=-309.546 z=481.128 mm, rx=2.7896 ry=1.107 rz=-0.2715 rad
      Waypoint Tip1_Lock: TCP in base x=-538.583 y=-338.869 z=236.944 mm, rx=0.0013 ry=-0.0083 rz=-2.1118 rad; joints [-137.124, -99.221, -76.057, -82.468, 93.606, 89.965] deg; pose in feature x=-139.482 y=-433.5 z=348.531 mm, rx=0.0139 ry=-0.0208 rz=-0.8958 rad; flange x=-488.924 y=-309.541 z=482.128 mm, rx=2.7896 ry=1.107 rz=-0.2715 rad
      Waypoint Tip1_Slip: TCP in base x=-538.568 y=-337.869 z=236.939 mm, rx=-0.0068 ry=0.0085 rz=3.1242 rad; joints [-131.488, -104.349, -68.619, -89.398, 80.899, 154.544] deg; pose in feature x=-140.414 y=-433.139 z=348.51 mm, rx=0.0255 ry=-0.0126 rz=-1.9429 rad; flange x=-490.024 y=-366.448 z=482.434 mm, rx=3.0718 ry=-0.4509 rz=-0.3328 rad
      Waypoint Tip1_high: TCP in base x=-538.968 y=-338.378 z=326.942 mm, rx=-0.0068 ry=0.0085 rz=3.1265 rad; joints [-131.445, -107.957, -50.262, -104.103, 80.885, 154.293] deg; pose in feature x=57.214 y=-30.744 z=76.425 mm, rx=0 ry=0.0001 rz=-2.0641 rad; flange x=-490.354 y=-366.84 z=572.437 mm, rx=3.0721 ry=-0.4473 rz=-0.3327 rad
  If New_tip≟4
    MoveL speed 250 mm/s, acceleration 1200 mm/s^2 (useActiveTCP=false) tcp=TCP_Tool1; feature=Joint_6_name
      Waypoint Tip2_High: TCP in base x=-538.644 y=-316.88 z=326.826 mm, rx=-0.0068 ry=0.0085 rz=3.1265 rad; joints [-132.848, -105.784, -53.248, -103.06, 81.079, 152.898] deg; pose in feature x=2.19 y=1.693 z=81.747 mm, rx=-0.0035 ry=0.0068 rz=-0.958 rad; flange x=-490.029 y=-345.343 z=572.321 mm, rx=3.0721 ry=-0.4473 rz=-0.3327 rad
      Waypoint Tip2_Press: TCP in base x=-538.255 y=-317.377 z=235.828 mm, rx=0.0012 ry=-0.0083 rz=-2.1095 rad; joints [-138.8, -97.629, -78.044, -82.173, 93.99, 88.199] deg; pose in feature x=-159.498 y=-425.724 z=347.078 mm, rx=0.0138 ry=-0.0208 rz=-0.8934 rad; flange x=-488.662 y=-287.93 z=481.011 mm, rx=2.7881 ry=1.1102 rz=-0.2712 rad
      Waypoint Tip2_Lock: TCP in base x=-538.259 y=-317.372 z=236.828 mm, rx=0.0012 ry=-0.0083 rz=-2.1095 rad; joints [-138.801, -97.64, -77.885, -82.321, 93.99, 88.197] deg; pose in feature x=-159.522 y=-425.727 z=348.078 mm, rx=0.0138 ry=-0.0208 rz=-0.8934 rad; flange x=-488.666 y=-287.924 z=482.011 mm, rx=2.7881 ry=1.1102 rz=-0.2712 rad
      Waypoint Tip2_Slip: TCP in base x=-538.244 y=-316.372 z=236.823 mm, rx=-0.0068 ry=0.0085 rz=3.1265 rad; joints [-132.898, -102.409, -71.128, -88.573, 81.109, 153.006] deg; pose in feature x=-160.454 y=-425.366 z=348.057 mm, rx=0.0255 ry=-0.0126 rz=-1.9406 rad; flange x=-489.629 y=-344.835 z=482.318 mm, rx=3.0721 ry=-0.4473 rz=-0.3327 rad
      Waypoint Tip2_High: TCP in base x=-538.644 y=-316.88 z=326.826 mm, rx=-0.0068 ry=0.0085 rz=3.1265 rad; joints [-132.848, -105.784, -53.248, -103.06, 81.079, 152.898] deg; pose in feature x=2.19 y=1.693 z=81.747 mm, rx=-0.0035 ry=0.0068 rz=-0.958 rad; flange x=-490.029 y=-345.343 z=572.321 mm, rx=3.0721 ry=-0.4473 rz=-0.3327 rad
  If New_tip≟5
    MoveL speed 250 mm/s, acceleration 1200 mm/s^2 (useActiveTCP=false) tcp=TCP_Tool1; feature=Joint_6_name
      Waypoint Tip3_High: TCP in base x=-538.312 y=-294.883 z=326.707 mm, rx=-0.0068 ry=0.0085 rz=3.1265 rad; joints [-134.359, -103.714, -56.012, -102.124, 81.293, 151.396] deg; pose in feature x=13.69 y=-3.755 z=-38.348 mm, rx=-0.1637 ry=0.1574 rz=-0.0025 rad; flange x=-489.697 y=-323.346 z=572.202 mm, rx=3.0721 ry=-0.4473 rz=-0.3327 rad
      Waypoint Tip3_Press: TCP in base x=-537.923 y=-295.38 z=235.709 mm, rx=0.0012 ry=-0.0083 rz=-2.1095 rad; joints [-140.579, -96.109, -79.753, -82.094, 94.365, 86.46] deg; pose in feature x=-180.005 y=-417.77 z=346.615 mm, rx=0.0138 ry=-0.0208 rz=-0.8934 rad; flange x=-488.33 y=-265.932 z=480.892 mm, rx=2.7881 ry=1.1102 rz=-0.2712 rad
      Waypoint Tip3_Lock: TCP in base x=-537.927 y=-295.375 z=236.709 mm, rx=0.0012 ry=-0.0083 rz=-2.1095 rad; joints [-140.58, -96.119, -79.595, -82.242, 94.365, 86.458] deg; pose in feature x=-180.029 y=-417.773 z=347.614 mm, rx=0.0138 ry=-0.0208 rz=-0.8934 rad; flange x=-488.334 y=-265.927 z=481.892 mm, rx=2.7881 ry=1.1102 rz=-0.2712 rad
      Waypoint Tip3_Slip: TCP in base x=-537.912 y=-294.375 z=236.704 mm, rx=-0.0068 ry=0.0085 rz=3.1265 rad; joints [-134.411, -100.547, -73.471, -87.848, 81.321, 151.499] deg; pose in feature x=-180.961 y=-417.412 z=347.593 mm, rx=0.0255 ry=-0.0126 rz=-1.9406 rad; flange x=-489.297 y=-322.838 z=482.199 mm, rx=3.0721 ry=-0.4473 rz=-0.3327 rad
      Waypoint Tip3_High: TCP in base x=-538.312 y=-294.883 z=326.707 mm, rx=-0.0068 ry=0.0085 rz=3.1265 rad; joints [-134.359, -103.714, -56.012, -102.124, 81.293, 151.396] deg; pose in feature x=13.69 y=-3.755 z=-38.348 mm, rx=-0.1637 ry=0.1574 rz=-0.0025 rad; flange x=-489.697 y=-323.346 z=572.202 mm, rx=3.0721 ry=-0.4473 rz=-0.3327 rad
  If New_tip≟6
    MoveL speed 250 mm/s, acceleration 1200 mm/s^2 (useActiveTCP=false) tcp=TCP_Tool1; feature=Joint_6_name
      Waypoint Tip4_High: TCP in base x=-537.988 y=-273.386 z=326.591 mm, rx=-0.0068 ry=0.0085 rz=3.1265 rad; joints [-135.913, -101.826, -58.462, -101.318, 81.519, 149.851] deg; pose in feature x=-0.038 y=0.033 z=76.429 mm, rx=0 ry=0.0001 rz=-2.0641 rad; flange x=-489.373 y=-301.849 z=572.086 mm, rx=3.0721 ry=-0.4473 rz=-0.3327 rad
      Waypoint Tip4_Press: TCP in base x=-537.598 y=-273.883 z=235.593 mm, rx=0.0012 ry=-0.0083 rz=-2.1095 rad; joints [-142.401, -94.722, -81.27, -82.089, 94.744, 84.678] deg; pose in feature x=-200.045 y=-409.997 z=346.162 mm, rx=0.0138 ry=-0.0208 rz=-0.8934 rad; flange x=-488.005 y=-244.435 z=480.776 mm, rx=2.7881 ry=1.1102 rz=-0.2712 rad
      Waypoint Tip4_Lock: TCP in base x=-537.603 y=-273.877 z=236.593 mm, rx=0.0012 ry=-0.0083 rz=-2.1095 rad; joints [-142.401, -94.732, -81.112, -82.237, 94.745, 84.676] deg; pose in feature x=-200.069 y=-410 z=347.161 mm, rx=0.0138 ry=-0.0208 rz=-0.8934 rad; flange x=-488.01 y=-244.43 z=481.776 mm, rx=2.7881 ry=1.1102 rz=-0.2712 rad
      Waypoint Tip4_Slip: TCP in base x=-537.588 y=-272.878 z=236.588 mm, rx=-0.0068 ry=0.0085 rz=3.1265 rad; joints [-135.967, -98.824, -75.586, -87.211, 81.546, 149.951] deg; pose in feature x=-201.001 y=-409.638 z=347.14 mm, rx=0.0255 ry=-0.0126 rz=-1.9406 rad; flange x=-488.973 y=-301.34 z=482.083 mm, rx=3.0721 ry=-0.4473 rz=-0.3327 rad
      Waypoint Tip4_High: TCP in base x=-537.988 y=-273.386 z=326.591 mm, rx=-0.0068 ry=0.0085 rz=3.1265 rad; joints [-135.913, -101.826, -58.462, -101.318, 81.519, 149.851] deg; pose in feature x=-0.038 y=0.033 z=76.429 mm, rx=0 ry=0.0001 rz=-2.0641 rad; flange x=-489.373 y=-301.849 z=572.086 mm, rx=3.0721 ry=-0.4473 rz=-0.3327 rad
  MoveJ speed 60 deg/s, acceleration 80 deg/s^2 (useActiveTCP=false) tcp=TCP_Tool1
    Waypoint Tip_change: TCP in base x=-81.571 y=-272.848 z=299.256 mm, rx=0 ry=0.0001 rz=-1.545 rad; joints [-70.556, -50.466, -101.854, -104.569, 84.569, 123.199] deg; flange x=-49.667 y=-215.719 z=542.134 mm, rx=2.3303 ry=1.8037 rz=-0.2542 rad
  If New_tip≠0
    Set NoAction tcp=TCP_Tips
  Old_tip := New_tip
SubProgram tool_change_JF (keepSynchronizedWithDisk=true trackProgramExecution=true) programFile=/programs/tool_change_JF.urp
  MoveJ speed 60 deg/s, acceleration 80 deg/s^2 (useActiveTCP=false) tcp=TCP_Schunk
    Waypoint Tool_change: TCP in base x=75.984 y=-313.148 z=341.083 mm, rx=0 ry=0.0001 rz=-0.2764 rad; joints [-56.431, -64.397, -114.786, -90.868, 90.559, 49.445] deg; flange x=75.993 y=-313.149 z=397.063 mm, rx=-0.4326 ry=-3.1115 rz=0 rad
  Set NoAction tcp=TCP_Schunk
  If Old_Tool≟1
    If Tool1≟ False
      MoveL speed 250 mm/s, acceleration 1200 mm/s^2 (useActiveTCP=false) tcp=TCP_Schunk; feature=Base
        Waypoint Tool_1_safe: TCP in base x=-227.333 y=-476.653 z=81.63 mm, rx=0.0068 ry=0.0007 rz=-0.2531 rad; joints [-103.501, -109.067, -114.718, -46.64, 90.288, 1.376] deg; flange x=-227.336 y=-477.036 z=137.608 mm, rx=-0.3963 ry=-3.1157 rz=-0.0106 rad
        Waypoint Tool1_on: TCP in base x=-376.178 y=-474.572 z=76.626 mm, rx=0.0067 ry=0.0008 rz=-0.2532 rad; joints [-117.914, -117.909, -101.757, -50.724, 90.219, -13.088] deg; flange x=-376.178 y=-474.953 z=132.605 mm, rx=-0.3964 ry=-3.1156 rz=-0.0106 rad
        Waypoint tool_1: TCP in base x=-376.117 y=-474.426 z=51.327 mm, rx=0.0068 ry=0.0008 rz=-0.2813 rad; joints [-117.918, -120.188, -102.793, -47.413, 90.203, -11.459] deg; flange x=-376.123 y=-474.809 z=107.305 mm, rx=-0.4402 ry=-3.1097 rz=-0.0106 rad
      Set DigitalOutput pin=digital_out[6]; digitalValue=0
      Set DigitalOutput (payload=0.78 tcpAsCog=false) tcp=TCP_Schunk; pin=digital_out[7]; digitalValue=1
      Wait Sleep waitTime=0.5
      Set DigitalOutput pin=digital_out[7]; digitalValue=0
      MoveL speed 250 mm/s, acceleration 1200 mm/s^2 (useActiveTCP=false) tcp=TCP_Schunk; feature=Base
        Waypoint Tool1_on: TCP in base x=-376.178 y=-474.572 z=76.626 mm, rx=0.0067 ry=0.0008 rz=-0.2532 rad; joints [-117.914, -117.909, -101.757, -50.724, 90.219, -13.088] deg; flange x=-376.178 y=-474.953 z=132.605 mm, rx=-0.3964 ry=-3.1156 rz=-0.0106 rad
    Else 
      Popup Message (haltProgram=false message=something blocking tool 1 storage inputType=Text)
  'skipping tool 0-> No tool on robot'
  If Old_Tool≟2
    If Tool2≟ False
      MoveL speed 250 mm/s, acceleration 1200 mm/s^2 (useActiveTCP=false) tcp=TCP_Schunk; feature=Base
        Waypoint Tool_2_safe: TCP in base x=-223.878 y=-311.698 z=82.74 mm, rx=0.0071 ry=0.0008 rz=-0.2532 rad; joints [-109.097, -91.747, -136.674, -42.016, 90.222, -4.143] deg; flange x=-223.881 y=-312.102 z=138.719 mm, rx=-0.3964 ry=-3.1156 rz=-0.0112 rad
        Waypoint tool2_on: TCP in base x=-373.864 y=-309.584 z=77.743 mm, rx=0.0071 ry=0.0007 rz=-0.2531 rad; joints [-127.272, -104.754, -121.779, -43.843, 90.117, -22.366] deg; flange x=-373.871 y=-309.984 z=133.721 mm, rx=-0.3963 ry=-3.1157 rz=-0.0111 rad
        Waypoint tool_2: TCP in base x=-373.87 y=-309.418 z=52.275 mm, rx=0.0069 ry=0.0008 rz=-0.2766 rad; joints [-127.289, -107.78, -122.985, -39.603, 90.088, -21.011] deg; flange x=-373.875 y=-309.809 z=108.254 mm, rx=-0.4329 ry=-3.1107 rz=-0.0109 rad
      Set DigitalOutput pin=digital_out[6]; digitalValue=0
      Set DigitalOutput (payload=0.78 tcpAsCog=false) tcp=TCP_Schunk; pin=digital_out[7]; digitalValue=1
      Wait Sleep waitTime=0.5
      Set DigitalOutput pin=digital_out[7]; digitalValue=0
      MoveL speed 250 mm/s, acceleration 1200 mm/s^2 (useActiveTCP=false) tcp=TCP_Schunk; feature=Base
        Waypoint tool2_on: TCP in base x=-373.864 y=-309.584 z=77.743 mm, rx=0.0071 ry=0.0007 rz=-0.2531 rad; joints [-127.272, -104.754, -121.779, -43.843, 90.117, -22.366] deg; flange x=-373.871 y=-309.984 z=133.721 mm, rx=-0.3963 ry=-3.1157 rz=-0.0111 rad
    Else 
      Popup Message (haltProgram=false message=something blocking tool 2 inputType=Text)
  If Old_Tool≟3
    If Tool3≟ False
      MoveL speed 250 mm/s, acceleration 1200 mm/s^2 (useActiveTCP=false) tcp=TCP_Schunk; feature=Base
        Waypoint Tool_3_safe: TCP in base x=-221.626 y=-146.719 z=83.867 mm, rx=0.0071 ry=0.0008 rz=-0.2532 rad; joints [-122.112, -71.21, -152.288, -46.895, 90.2, -17.154] deg; flange x=-221.627 y=-147.119 z=139.846 mm, rx=-0.3964 ry=-3.1156 rz=-0.0111 rad
        Waypoint tool_3_on: TCP in base x=-371.646 y=-144.64 z=78.859 mm, rx=0.0071 ry=0.0007 rz=-0.2532 rad; joints [-142.715, -94.273, -134.837, -41.189, 90.022, -37.761] deg; flange x=-371.65 y=-145.041 z=134.838 mm, rx=-0.3964 ry=-3.1156 rz=-0.0112 rad
        Waypoint tool_3: TCP in base x=-371.626 y=-144.442 z=53.376 mm, rx=0.0071 ry=0.0007 rz=-0.2532 rad; joints [-142.741, -98.093, -136.292, -35.914, 89.98, -37.755] deg; flange x=-371.631 y=-144.842 z=109.354 mm, rx=-0.3965 ry=-3.1156 rz=-0.0111 rad
      Set DigitalOutput pin=digital_out[6]; digitalValue=0
      Set DigitalOutput (payload=0.78 tcpAsCog=false) tcp=TCP_Schunk; pin=digital_out[7]; digitalValue=1
      Wait Sleep waitTime=0.5
      Set DigitalOutput pin=digital_out[7]; digitalValue=0
      MoveL speed 250 mm/s, acceleration 1200 mm/s^2 (useActiveTCP=true) feature=Base
        Waypoint tool_3_on: TCP in base x=-371.646 y=-144.64 z=78.859 mm, rx=0.0071 ry=0.0007 rz=-0.2532 rad; joints [-142.715, -94.273, -134.837, -41.189, 90.022, -37.761] deg; flange x=-371.65 y=-145.041 z=134.838 mm, rx=-0.3964 ry=-3.1156 rz=-0.0112 rad
    Else 
      Popup Message (haltProgram=false message=something blocking tool3 storage inputType=Text)
  If New_Tool≟1
    If Tool1≟ True
      MoveL speed 250 mm/s, acceleration 1200 mm/s^2 (useActiveTCP=false) tcp=TCP_Schunk; feature=Base
        Waypoint Tool1_on: TCP in base x=-376.178 y=-474.572 z=76.626 mm, rx=0.0067 ry=0.0008 rz=-0.2532 rad; joints [-117.914, -117.909, -101.757, -50.724, 90.219, -13.088] deg; flange x=-376.178 y=-474.953 z=132.605 mm, rx=-0.3964 ry=-3.1156 rz=-0.0106 rad
        Waypoint tool_1: TCP in base x=-376.117 y=-474.426 z=51.327 mm, rx=0.0068 ry=0.0008 rz=-0.2813 rad; joints [-117.918, -120.188, -102.793, -47.413, 90.203, -11.459] deg; flange x=-376.123 y=-474.809 z=107.305 mm, rx=-0.4402 ry=-3.1097 rz=-0.0106 rad
      Set DigitalOutput (payload=1.41 tcpAsCog=false) tcp=TCP_Tool1; pin=digital_out[6]; digitalValue=1
      Wait Sleep waitTime=0.5
      MoveL speed 250 mm/s, acceleration 1200 mm/s^2 (useActiveTCP=false) tcp=TCP_Schunk; feature=Base
        Waypoint Tool1_on: TCP in base x=-376.178 y=-474.572 z=76.626 mm, rx=0.0067 ry=0.0008 rz=-0.2532 rad; joints [-117.914, -117.909, -101.757, -50.724, 90.219, -13.088] deg; flange x=-376.178 y=-474.953 z=132.605 mm, rx=-0.3964 ry=-3.1156 rz=-0.0106 rad
        Waypoint Tool_1_safe: TCP in base x=-227.333 y=-476.653 z=81.63 mm, rx=0.0068 ry=0.0007 rz=-0.2531 rad; joints [-103.501, -109.067, -114.718, -46.64, 90.288, 1.376] deg; flange x=-227.336 y=-477.036 z=137.608 mm, rx=-0.3963 ry=-3.1157 rz=-0.0106 rad
    Else 
      Popup Message (haltProgram=false message=tool 1 not in place inputType=Text)
  If New_Tool≟2
    If Tool2≟ True
      MoveL speed 250 mm/s, acceleration 1200 mm/s^2 (useActiveTCP=false) tcp=TCP_Schunk; feature=Base
        Waypoint tool2_on: TCP in base x=-373.864 y=-309.584 z=77.743 mm, rx=0.0071 ry=0.0007 rz=-0.2531 rad; joints [-127.272, -104.754, -121.779, -43.843, 90.117, -22.366] deg; flange x=-373.871 y=-309.984 z=133.721 mm, rx=-0.3963 ry=-3.1157 rz=-0.0111 rad
        Waypoint tool_2: TCP in base x=-373.87 y=-309.418 z=52.275 mm, rx=0.0069 ry=0.0008 rz=-0.2766 rad; joints [-127.289, -107.78, -122.985, -39.603, 90.088, -21.011] deg; flange x=-373.875 y=-309.809 z=108.254 mm, rx=-0.4329 ry=-3.1107 rz=-0.0109 rad
      Set DigitalOutput (payload=1.87 tcpAsCog=false) tcp=TCP_Tool2; pin=digital_out[6]; digitalValue=1
      Set SingleDigitalPulseActionState SingleDigitalPulseActionState(hiPulseInSeconds=0.5, pin=digital_out[0])
      Wait Sleep waitTime=0.5
      MoveL speed 250 mm/s, acceleration 1200 mm/s^2 (useActiveTCP=false) tcp=TCP_Schunk; feature=Base
        Waypoint tool2_on: TCP in base x=-373.864 y=-309.584 z=77.743 mm, rx=0.0071 ry=0.0007 rz=-0.2531 rad; joints [-127.272, -104.754, -121.779, -43.843, 90.117, -22.366] deg; flange x=-373.871 y=-309.984 z=133.721 mm, rx=-0.3963 ry=-3.1157 rz=-0.0111 rad
        Waypoint Tool_2_safe: TCP in base x=-223.878 y=-311.698 z=82.74 mm, rx=0.0071 ry=0.0008 rz=-0.2532 rad; joints [-109.097, -91.747, -136.674, -42.016, 90.222, -4.143] deg; flange x=-223.881 y=-312.102 z=138.719 mm, rx=-0.3964 ry=-3.1156 rz=-0.0112 rad
    Else 
      Popup Message (haltProgram=false message=tool 2 not in place inputType=Text)
  If New_Tool≟3
    If Tool3≟ True
      MoveL speed 250 mm/s, acceleration 1200 mm/s^2 (useActiveTCP=false) tcp=TCP_Schunk; feature=Base
        Waypoint tool_3_on: TCP in base x=-371.646 y=-144.64 z=78.859 mm, rx=0.0071 ry=0.0007 rz=-0.2532 rad; joints [-142.715, -94.273, -134.837, -41.189, 90.022, -37.761] deg; flange x=-371.65 y=-145.041 z=134.838 mm, rx=-0.3964 ry=-3.1156 rz=-0.0112 rad
        Waypoint tool_3: TCP in base x=-371.626 y=-144.442 z=53.376 mm, rx=0.0071 ry=0.0007 rz=-0.2532 rad; joints [-142.741, -98.093, -136.292, -35.914, 89.98, -37.755] deg; flange x=-371.631 y=-144.842 z=109.354 mm, rx=-0.3965 ry=-3.1156 rz=-0.0111 rad
      Set DigitalOutput (payload=1.28 tcpAsCog=false) tcp=TCP_Tool3; pin=digital_out[6]; digitalValue=1
      Wait Sleep waitTime=0.5
      MoveL speed 250 mm/s, acceleration 1200 mm/s^2 (useActiveTCP=false) tcp=TCP_Schunk; feature=Base
        Waypoint tool_3_on: TCP in base x=-371.646 y=-144.64 z=78.859 mm, rx=0.0071 ry=0.0007 rz=-0.2532 rad; joints [-142.715, -94.273, -134.837, -41.189, 90.022, -37.761] deg; flange x=-371.65 y=-145.041 z=134.838 mm, rx=-0.3964 ry=-3.1156 rz=-0.0112 rad
        Waypoint Tool_3_safe: TCP in base x=-221.626 y=-146.719 z=83.867 mm, rx=0.0071 ry=0.0008 rz=-0.2532 rad; joints [-122.112, -71.21, -152.288, -46.895, 90.2, -17.154] deg; flange x=-221.627 y=-147.119 z=139.846 mm, rx=-0.3964 ry=-3.1156 rz=-0.0111 rad
    Else 
      Popup Message (haltProgram=false message=tool  3 not in place inputType=Text)
  MoveJ speed 60 deg/s, acceleration 80 deg/s^2 (useActiveTCP=true)
    Waypoint Tool_change: TCP in base x=75.984 y=-313.148 z=341.083 mm, rx=0 ry=0.0001 rz=-0.2764 rad; joints [-56.431, -64.397, -114.786, -90.868, 90.559, 49.445] deg; flange x=75.993 y=-313.149 z=397.063 mm, rx=-0.4326 ry=-3.1115 rz=0 rad
  Old_Tool := New_Tool
